{attribute 'pack_mode' := '1'}  // needed for python pyads reading
TYPE ST_ComOut_ExportStation :
STRUCT
	Enable: BOOL;
	ProcessComplete: BOOL;
	OK: BOOL;
	NOK: BOOL;
	Error: BOOL;
	StatusWord: INT;
	StationName: INT;
	Error_ID: INT;
	ProcesedMover: STRING(13);
	MoversList: ARRAY[1..10] OF STRING(13);
END_STRUCT
END_TYPE

(* stored: Version 1.1.0.1
   DUT ST_ComOut_ExportStation: Id {440a6a1e-a622-4120-9f4b-71ed55d22c06} *)
